(* IEC 61131-3 sources: SRCI/RobotLibrary/Library/Functions/Convert/TO_STRING (part 3) *)

(* ---- TELEGRAM_STATE_TO_STRING.st ---- *)
FUNCTION TELEGRAM_STATE_TO_STRING : STRING
// -------------------------------------------------------------------------
//  SRCI Robot Library
// -------------------------------------------------------------------------
//
//  Object:      TelegramStateToString
//  Author:      Thorsten Brach
//  Date:        2024-11-16
//
//  Description:
//
//
//  Copyright:
//    (C) 2024 Thorsten Brach. All rights reserved
//             Licensed under the LGPL-3.0 license.
//
//  Disclaimer:
//    This project is provided without any guarantee and can be used for
//    private and commercial purposes. Any use is at the user’s
//    own risk and responsibility.
//
// -------------------------------------------------------------------------
VAR_INPUT
  /// Telegram state
  State : TelegramState;
END_VAR

  CASE State
  OF
    TelegramState.UNDEFINED                : TELEGRAM_STATE_TO_STRING := StrReplace('UNDEFINED ({0})'               ,'{0}', USINT_TO_STRING(State));
    TelegramState.ERROR_161                : TELEGRAM_STATE_TO_STRING := StrReplace('ERROR_161 ({0})'               ,'{0}', USINT_TO_STRING(State));
    TelegramState.ERROR_162                : TELEGRAM_STATE_TO_STRING := StrReplace('ERROR_162 ({0})'               ,'{0}', USINT_TO_STRING(State));
    TelegramState.ERROR_163                : TELEGRAM_STATE_TO_STRING := StrReplace('ERROR_163 ({0})'               ,'{0}', USINT_TO_STRING(State));
    TelegramState.ERROR_164                : TELEGRAM_STATE_TO_STRING := StrReplace('ERROR_164 ({0})'               ,'{0}', USINT_TO_STRING(State));
    TelegramState.ERROR_165                : TELEGRAM_STATE_TO_STRING := StrReplace('ERROR_165 ({0})'               ,'{0}', USINT_TO_STRING(State));
    TelegramState.ERROR_166                : TELEGRAM_STATE_TO_STRING := StrReplace('ERROR_166 ({0})'               ,'{0}', USINT_TO_STRING(State));
    TelegramState.ERROR_167                : TELEGRAM_STATE_TO_STRING := StrReplace('ERROR_167 ({0})'               ,'{0}', USINT_TO_STRING(State));
    TelegramState.ERROR_168                : TELEGRAM_STATE_TO_STRING := StrReplace('ERROR_168 ({0})'               ,'{0}', USINT_TO_STRING(State));
    TelegramState.ERROR_169                : TELEGRAM_STATE_TO_STRING := StrReplace('ERROR_169 ({0})'               ,'{0}', USINT_TO_STRING(State));
    TelegramState.ERROR_170                : TELEGRAM_STATE_TO_STRING := StrReplace('ERROR_170 ({0})'               ,'{0}', USINT_TO_STRING(State));
    TelegramState.ERROR_171                : TELEGRAM_STATE_TO_STRING := StrReplace('ERROR_171 ({0})'               ,'{0}', USINT_TO_STRING(State));
    TelegramState.ERROR_172                : TELEGRAM_STATE_TO_STRING := StrReplace('ERROR_172 ({0})'               ,'{0}', USINT_TO_STRING(State));
    TelegramState.ERROR_173                : TELEGRAM_STATE_TO_STRING := StrReplace('ERROR_173 ({0})'               ,'{0}', USINT_TO_STRING(State));
    TelegramState.READY_TO_RESUME          : TELEGRAM_STATE_TO_STRING := StrReplace('READY_TO_RESUME ({0})'         ,'{0}', USINT_TO_STRING(State));
    TelegramState.READY_FOR_INITIALIZATION : TELEGRAM_STATE_TO_STRING := StrReplace('READY_FOR_INITIALIZATION ({0})','{0}', USINT_TO_STRING(State));
    TelegramState.INITIALIZED              : TELEGRAM_STATE_TO_STRING := StrReplace('INITIALIZED ({0})'             ,'{0}', USINT_TO_STRING(State));
  ELSE
    TELEGRAM_STATE_TO_STRING := CONCAT('TELEGRAM_STATE_TO_STRING Function: Error -> no parsing for value ', USINT_TO_STRING(State));
  END_CASE

END_FUNCTION

(* ---- THRESHOLD_MODE_TO_STRING.st ---- *)
FUNCTION THRESHOLD_MODE_TO_STRING : STRING
// -------------------------------------------------------------------------
//  SRCI Robot Library
// -------------------------------------------------------------------------
//
//  Object:      THRESHOLD_MODE_TO_STRING
//  Author:      Thorsten Brach
//  Date:        2025-01-24
//
//  Description:
//
//
//  Copyright:
//    (C) 2025 Thorsten Brach. All rights reserved
//             Licensed under the LGPL-3.0 license.
//
//  Disclaimer:
//    This project is provided without any guarantee and can be used for
//    private and commercial purposes. Any use is at the user’s
//    own risk and responsibility.
//
// -------------------------------------------------------------------------
VAR_INPUT
  /// ThresholdMode
  Value : ThresholdMode;
END_VAR

  CASE Value
  OF
    ThresholdMode.AUTOMATIC : THRESHOLD_MODE_TO_STRING := StrReplace('AUTOMATIC ({0})','{0}' , USINT_TO_STRING(Value));
    ThresholdMode.MANUAL    : THRESHOLD_MODE_TO_STRING := StrReplace('MANUAL ({0})'   ,'{0}' , USINT_TO_STRING(Value));
  ELSE
    THRESHOLD_MODE_TO_STRING := CONCAT('THRESHOLD_MODE_TO_STRING Function: Error -> no parsing for value ', USINT_TO_STRING(Value));
  END_CASE

END_FUNCTION

(* ---- TOOL_CALCULATION_MODE_TO_STRING.st ---- *)
FUNCTION TOOL_CALCULATION_MODE_TO_STRING : STRING
// -------------------------------------------------------------------------
//  SRCI Robot Library
// -------------------------------------------------------------------------
//
//  Object:      TOOL_CALCULATION_MODE_TO_STRING
//  Author:      Thorsten Brach
//  Date:        2025-02-01
//
//  Description:
//
//
//  Copyright:
//    (C) 2025 Thorsten Brach. All rights reserved
//             Licensed under the LGPL-3.0 license.
//
//  Disclaimer:
//    This project is provided without any guarantee and can be used for
//    private and commercial purposes. Any use is at the user’s
//    own risk and responsibility.
//
// -------------------------------------------------------------------------
VAR_INPUT
  /// ToolCalculationMode
  Value : ToolCalculationMode;
END_VAR

  CASE Value
  OF
    ToolCalculationMode.TWO_POINT_Z_METHOD   : TOOL_CALCULATION_MODE_TO_STRING := StrReplace('TWO_POINT_Z_METHOD ({0})'  ,'{0}' , SINT_TO_STRING(Value));
    ToolCalculationMode.THREE_POINT_METHOD   : TOOL_CALCULATION_MODE_TO_STRING := StrReplace('THREE_POINT_METHOD ({0})'  ,'{0}' , SINT_TO_STRING(Value));
    ToolCalculationMode.FOUR_POINT_METHOD    : TOOL_CALCULATION_MODE_TO_STRING := StrReplace('FOUR_POINT_METHOD ({0})'   ,'{0}' , SINT_TO_STRING(Value));
    ToolCalculationMode.FIVE_POINT_METHOD    : TOOL_CALCULATION_MODE_TO_STRING := StrReplace('FIVE_POINT_METHOD ({0})'   ,'{0}' , SINT_TO_STRING(Value));
    ToolCalculationMode.SIX_POINT_METHOD     : TOOL_CALCULATION_MODE_TO_STRING := StrReplace('SIX_POINT_METHOD ({0})'    ,'{0}' , SINT_TO_STRING(Value));
    ToolCalculationMode.ABC_WORLD_METHOD     : TOOL_CALCULATION_MODE_TO_STRING := StrReplace('ABC_WORLD_METHOD ({0})'    ,'{0}' , SINT_TO_STRING(Value));
    ToolCalculationMode.ABC_TWO_POINT_METHOD : TOOL_CALCULATION_MODE_TO_STRING := StrReplace('ABC_TWO_POINT_METHOD ({0})','{0}' , SINT_TO_STRING(Value));
  ELSE
    TOOL_CALCULATION_MODE_TO_STRING := CONCAT('TOOL_CALCULATION_MODE_TO_STRING Function: Error -> no parsing for value ', SINT_TO_STRING(Value));
  END_CASE

END_FUNCTION

(* ---- TRAJECTORY_MODE_TO_STRING.st ---- *)
FUNCTION TRAJECTORY_MODE_TO_STRING : STRING
// -------------------------------------------------------------------------
//  SRCI Robot Library
// -------------------------------------------------------------------------
//
//  Object:      TRAJECTORY_MODE_TO_STRING
//  Author:      Thorsten Brach
//  Date:        2025-03-01
//
//  Description:
//
//
//  Copyright:
//    (C) 2025 Thorsten Brach. All rights reserved
//             Licensed under the LGPL-3.0 license.
//
//  Disclaimer:
//    This project is provided without any guarantee and can be used for
//    private and commercial purposes. Any use is at the user’s
//    own risk and responsibility.
//
// -------------------------------------------------------------------------
VAR_INPUT
  /// TrajectoryMode
  Value : TrajectoryMode;
END_VAR

  CASE Value
  OF
    TrajectoryMode.INVALID          : TRAJECTORY_MODE_TO_STRING := StrReplace('INVALID ({0})'         ,'{0}' , USINT_TO_STRING(Value));
    TrajectoryMode.LINEAR_MOVEMENT  : TRAJECTORY_MODE_TO_STRING := StrReplace('LINEAR_MOVEMENT ({0})' ,'{0}' , USINT_TO_STRING(Value));
    TrajectoryMode.PTP_MOVEMENT     : TRAJECTORY_MODE_TO_STRING := StrReplace('PTP_MOVEMENT ({0})'    ,'{0}' , USINT_TO_STRING(Value));
  ELSE
    TRAJECTORY_MODE_TO_STRING := CONCAT('TRAJECTORY_MODE_TO_STRING Function: Error -> no parsing for value ', USINT_TO_STRING(Value));
  END_CASE

END_FUNCTION

(* ---- TRANSFORM_MODE_TO_STRING.st ---- *)
FUNCTION TRANSFORM_MODE_TO_STRING : STRING
// -------------------------------------------------------------------------
//  SRCI Robot Library
// -------------------------------------------------------------------------
//
//  Object:      TRANSFORM_MODE_TO_STRING
//  Author:      Thorsten Brach
//  Date:        2025-01-24
//
//  Description:
//
//
//  Copyright:
//    (C) 2025 Thorsten Brach. All rights reserved
//             Licensed under the LGPL-3.0 license.
//
//  Disclaimer:
//    This project is provided without any guarantee and can be used for
//    private and commercial purposes. Any use is at the user’s
//    own risk and responsibility.
//
// -------------------------------------------------------------------------
VAR_INPUT
  /// TransformMode
  Value : TransformMode;
END_VAR

  CASE Value
  OF
    TransformMode.MIRROR_AT_POINT             : TRANSFORM_MODE_TO_STRING := StrReplace('MIRROR_AT_POINT ({0})'             ,'{0}' , SINT_TO_STRING(Value));
    TransformMode.MIRROR_AT_STRAIGHT_LINE     : TRANSFORM_MODE_TO_STRING := StrReplace('MIRROR_AT_STRAIGHT_LINE ({0})'     ,'{0}' , SINT_TO_STRING(Value));
    TransformMode.MIRROR_AT_PLANE             : TRANSFORM_MODE_TO_STRING := StrReplace('MIRROR_AT_PLANE ({0})'             ,'{0}' , SINT_TO_STRING(Value));
    TransformMode.ROTATE_AROUND_STRAIGHT_LINE : TRANSFORM_MODE_TO_STRING := StrReplace('ROTATE_AROUND_STRAIGHT_LINE ({0})' ,'{0}' , SINT_TO_STRING(Value));
    TransformMode.SHIFT_BY_VECTOR             : TRANSFORM_MODE_TO_STRING := StrReplace('SHIFT_BY_VECTOR ({0})'             ,'{0}' , SINT_TO_STRING(Value));
  ELSE
    TRANSFORM_MODE_TO_STRING := CONCAT('TRANSFORM_MODE_TO_STRING Function: Error -> no parsing for value ', SINT_TO_STRING(Value));
  END_CASE

END_FUNCTION

(* ---- TRIGGER_CONDITION_TO_STRING.st ---- *)
FUNCTION TRIGGER_CONDITION_TO_STRING : STRING
// -------------------------------------------------------------------------
//  SRCI Robot Library
// -------------------------------------------------------------------------
//
//  Object:      TRIGGER_CONDITION_TO_STRING
//  Author:      Thorsten Brach
//  Date:        2025-02-01
//
//  Description:
//
//
//  Copyright:
//    (C) 2025 Thorsten Brach. All rights reserved
//             Licensed under the LGPL-3.0 license.
//
//  Disclaimer:
//    This project is provided without any guarantee and can be used for
//    private and commercial purposes. Any use is at the user’s
//    own risk and responsibility.
//
// -------------------------------------------------------------------------
VAR_INPUT
  /// TriggerCondition
  Value : TriggerCondition;
END_VAR

  CASE Value
  OF
    TriggerCondition.TARGET_POSITION_TIME_MS                : TRIGGER_CONDITION_TO_STRING := StrReplace('TARGET_POSITION_TIME_MS ({0})'               ,'{0}' , SINT_TO_STRING(Value));
    TriggerCondition.TARGET_POSITION_TCP_VELOCITY_ABSOLUTE  : TRIGGER_CONDITION_TO_STRING := StrReplace('TARGET_POSITION_TCP_VELOCITY_ABSOLUTE ({0})' ,'{0}' , SINT_TO_STRING(Value));
    TriggerCondition.TARGET_POSITION_TCP_VELOCITY_PERCENT   : TRIGGER_CONDITION_TO_STRING := StrReplace('TARGET_POSITION_TCP_VELOCITY_PERCENT ({0})'  ,'{0}' , SINT_TO_STRING(Value));
    TriggerCondition.TARGET_POSITION_DISTANCE_ABSOLUTE      : TRIGGER_CONDITION_TO_STRING := StrReplace('TARGET_POSITION_DISTANCE_ABSOLUTE ({0})'     ,'{0}' , SINT_TO_STRING(Value));
    TriggerCondition.TARGET_POSITION_DISTANCE_PERCENT       : TRIGGER_CONDITION_TO_STRING := StrReplace('TARGET_POSITION_DISTANCE_PERCENT ({0})'      ,'{0}' , SINT_TO_STRING(Value));
    TriggerCondition.UNDEFINED                              : TRIGGER_CONDITION_TO_STRING := StrReplace('UNDEFINED ({0})'                             ,'{0}' , SINT_TO_STRING(Value));
    TriggerCondition.START_POSITION_DISTANCE_PERCENT        : TRIGGER_CONDITION_TO_STRING := StrReplace('START_POSITION_DISTANCE_PERCENT ({0})'       ,'{0}' , SINT_TO_STRING(Value));
    TriggerCondition.START_POSITION_DISTANCE_ABSOLUTE       : TRIGGER_CONDITION_TO_STRING := StrReplace('START_POSITION_DISTANCE_ABSOLUTE ({0})'      ,'{0}' , SINT_TO_STRING(Value));
    TriggerCondition.START_POSITION_TCP_VELOCITY_PERCENT    : TRIGGER_CONDITION_TO_STRING := StrReplace('START_POSITION_TCP_VELOCITY_PERCENT ({0})'   ,'{0}' , SINT_TO_STRING(Value));
    TriggerCondition.START_POSITION_TCP_VELOCIT_ABSOLUTE    : TRIGGER_CONDITION_TO_STRING := StrReplace('START_POSITION_TCP_VELOCIT_ABSOLUTE ({0})'   ,'{0}' , SINT_TO_STRING(Value));
    TriggerCondition.START_POSITION_TIME_MS                 : TRIGGER_CONDITION_TO_STRING := StrReplace('START_POSITION_TCP_VELOCIT_ABSOLUTE ({0})'   ,'{0}' , SINT_TO_STRING(Value));
  ELSE
    TRIGGER_CONDITION_TO_STRING := CONCAT('TRIGGER_CONDITION_TO_STRING Function: Error -> no parsing for value ', SINT_TO_STRING(Value));
  END_CASE

END_FUNCTION

(* ---- TRIGGER_MODE_IO_TO_STRING.st ---- *)
FUNCTION TRIGGER_MODE_IO_TO_STRING : STRING
// -------------------------------------------------------------------------
//  SRCI Robot Library
// -------------------------------------------------------------------------
//
//  Object:      TRIGGER_MODE_IO_TO_STRING
//  Author:      Thorsten Brach
//  Date:        2025-02-01
//
//  Description:
//
//
//  Copyright:
//    (C) 2025 Thorsten Brach. All rights reserved
//             Licensed under the LGPL-3.0 license.
//
//  Disclaimer:
//    This project is provided without any guarantee and can be used for
//    private and commercial purposes. Any use is at the user’s
//    own risk and responsibility.
//
// -------------------------------------------------------------------------
VAR_INPUT
  /// TriggerModeIo
  Value : TriggerModeIo;
END_VAR

  CASE Value
  OF
    TriggerModeIo.INVALID                                                             : TRIGGER_MODE_IO_TO_STRING := StrReplace('INVALID ({0})'                                                              ,'{0}' , SINT_TO_STRING(Value));
    TriggerModeIo.DIGITAL_INPUT_RISING_EDGE                                           : TRIGGER_MODE_IO_TO_STRING := StrReplace('DIGITAL_INPUT_RISING_EDGE ({0})'                                            ,'{0}' , SINT_TO_STRING(Value));
    TriggerModeIo.DIGITAL_INPUT_FALLING_EDGE                                          : TRIGGER_MODE_IO_TO_STRING := StrReplace('DIGITAL_INPUT_FALLING_EDGE ({0})'                                           ,'{0}' , SINT_TO_STRING(Value));
    TriggerModeIo.DIGITAL_INPUT_RISING_OR_FALLING_EDGE                                : TRIGGER_MODE_IO_TO_STRING := StrReplace('DIGITAL_INPUT_RISING_OR_FALLING_EDGE ({0})'                                 ,'{0}' , SINT_TO_STRING(Value));
    TriggerModeIo.DIGITAL_INPUT_RISING_OR_FALLING_EDGE_INVERTED                       : TRIGGER_MODE_IO_TO_STRING := StrReplace('DIGITAL_INPUT_RISING_OR_FALLING_EDGE_INVERTED ({0})'                        ,'{0}' , SINT_TO_STRING(Value));
    TriggerModeIo.DIGITAL_OUTPUT_RISING_EDGE                                          : TRIGGER_MODE_IO_TO_STRING := StrReplace('DIGITAL_OUTPUT_RISING_EDGE ({0})'                                           ,'{0}' , SINT_TO_STRING(Value));
    TriggerModeIo.DIGITAL_OUTPUT_FALLING_EDGE                                         : TRIGGER_MODE_IO_TO_STRING := StrReplace('DIGITAL_OUTPUT_FALLING_EDGE ({0})'                                          ,'{0}' , SINT_TO_STRING(Value));
    TriggerModeIo.DIGITAL_OUTPUT_RISING_OR_FALLING_EDGE                               : TRIGGER_MODE_IO_TO_STRING := StrReplace('DIGITAL_OUTPUT_RISING_OR_FALLING_EDGE ({0})'                                ,'{0}' , SINT_TO_STRING(Value));
    TriggerModeIo.DIGITAL_OUTPUT_RISING_OR_FALLING_EDGE_INVERTED                      : TRIGGER_MODE_IO_TO_STRING := StrReplace('DIGITAL_OUTPUT_RISING_OR_FALLING_EDGE_INVERTED ({0})'                       ,'{0}' , SINT_TO_STRING(Value));
    TriggerModeIo.ANALOG_INPUT_EXCEEDING_DEFINED_THRESHOLD                            : TRIGGER_MODE_IO_TO_STRING := StrReplace('ANALOG_INPUT_EXCEEDING_DEFINED_THRESHOLD ({0})'                             ,'{0}' , SINT_TO_STRING(Value));
    TriggerModeIo.ANALOG_INPUT_FALLING_BELOW_DEFINED_THRESHOLD                        : TRIGGER_MODE_IO_TO_STRING := StrReplace('ANALOG_INPUT_FALLING_BELOW_DEFINED_THRESHOLD ({0})'                         ,'{0}' , SINT_TO_STRING(Value));
    TriggerModeIo.ANALOG_INPUT_EXCEEDING_OR_FALLING_BELOW_DEFINED_THRESHOLD           : TRIGGER_MODE_IO_TO_STRING := StrReplace('ANALOG_INPUT_EXCEEDING_OR_FALLING_BELOW_DEFINED_THRESHOLD ({0})'            ,'{0}' , SINT_TO_STRING(Value));
    TriggerModeIo.ANALOG_INPUT_EXCEEDING_OR_FALLING_BELOW_DEFINED_THRESHOLD_INVERTED  : TRIGGER_MODE_IO_TO_STRING := StrReplace('ANALOG_INPUT_EXCEEDING_OR_FALLING_BELOW_DEFINED_THRESHOLD_INVERTED ({0})'   ,'{0}' , SINT_TO_STRING(Value));
    TriggerModeIo.ANALOG_INPUT_ENTERING_DEFINED_RANGE                                 : TRIGGER_MODE_IO_TO_STRING := StrReplace('ANALOG_INPUT_ENTERING_DEFINED_RANGE ({0})'                                  ,'{0}' , SINT_TO_STRING(Value));
    TriggerModeIo.ANALOG_INPUT_LEAVING_DEFINED_RANGE                                  : TRIGGER_MODE_IO_TO_STRING := StrReplace('ANALOG_INPUT_LEAVING_DEFINED_RANGE ({0})'                                   ,'{0}' , SINT_TO_STRING(Value));
    TriggerModeIo.ANALOG_INPUT_ENTERING_OR_LEAVING_DEFINED_RANGE                      : TRIGGER_MODE_IO_TO_STRING := StrReplace('ANALOG_INPUT_ENTERING_OR_LEAVING_DEFINED_RANGE ({0})'                       ,'{0}' , SINT_TO_STRING(Value));
    TriggerModeIo.ANALOG_INPUT_ENTERING_OR_LEAVING_DEFINED_RANGE_INVERTED             : TRIGGER_MODE_IO_TO_STRING := StrReplace('ANALOG_INPUT_ENTERING_OR_LEAVING_DEFINED_RANGE_INVERTED ({0})'              ,'{0}' , SINT_TO_STRING(Value));
    TriggerModeIo.ANALOG_OUTPUT_EXCEEDING_DEFINED_THRESHOLD                           : TRIGGER_MODE_IO_TO_STRING := StrReplace('ANALOG_OUTPUT_EXCEEDING_DEFINED_THRESHOLD ({0})'                            ,'{0}' , SINT_TO_STRING(Value));
    TriggerModeIo.ANALOG_OUTPUT_FALLING_BELOW_DEFINED_THRESHOLD                       : TRIGGER_MODE_IO_TO_STRING := StrReplace('ANALOG_OUTPUT_FALLING_BELOW_DEFINED_THRESHOLD ({0})'                        ,'{0}' , SINT_TO_STRING(Value));
    TriggerModeIo.ANALOG_OUTPUT_EXCEEDING_OR_FALLING_BELOW_DEFINED_THRESHOLD          : TRIGGER_MODE_IO_TO_STRING := StrReplace('ANALOG_OUTPUT_EXCEEDING_OR_FALLING_BELOW_DEFINED_THRESHOLD ({0})'           ,'{0}' , SINT_TO_STRING(Value));
    TriggerModeIo.ANALOG_OUTPUT_EXCEEDING_OR_FALLING_BELOW_DEFINED_THRESHOLD_INVERTED : TRIGGER_MODE_IO_TO_STRING := StrReplace('ANALOG_OUTPUT_EXCEEDING_OR_FALLING_BELOW_DEFINED_THRESHOLD_INVERTED ({0})'  ,'{0}' , SINT_TO_STRING(Value));
    TriggerModeIo.ANALOG_OUTPUT_ENTERING_DEFINED_RANGE                                : TRIGGER_MODE_IO_TO_STRING := StrReplace('ANALOG_OUTPUT_ENTERING_DEFINED_RANGE ({0})'                                 ,'{0}' , SINT_TO_STRING(Value));
    TriggerModeIo.ANALOG_OUTPUT_LEAVING_DEFINED_RANGE                                 : TRIGGER_MODE_IO_TO_STRING := StrReplace('ANALOG_OUTPUT_LEAVING_DEFINED_RANGE ({0})'                                  ,'{0}' , SINT_TO_STRING(Value));
    TriggerModeIo.ANALOG_OUTPUT_ENTERING_OR_LEAVING_DEFINED_RANGE                     : TRIGGER_MODE_IO_TO_STRING := StrReplace('ANALOG_OUTPUT_ENTERING_OR_LEAVING_DEFINED_RANGE ({0})'                      ,'{0}' , SINT_TO_STRING(Value));
    TriggerModeIo.ANALOG_OUTPUT_ENTERING_OR_LEAVING_DEFINED_RANGE_INVERTED            : TRIGGER_MODE_IO_TO_STRING := StrReplace('ANALOG_OUTPUT_ENTERING_OR_LEAVING_DEFINED_RANGE_INVERTED ({0})'             ,'{0}' , SINT_TO_STRING(Value));
    TriggerModeIo.INTEGER_REGISTER_EXCEEDING_DEFINED_THRESHOLD                        : TRIGGER_MODE_IO_TO_STRING := StrReplace('INTEGER_REGISTER_EXCEEDING_DEFINED_THRESHOLD ({0})'                         ,'{0}' , SINT_TO_STRING(Value));
    TriggerModeIo.INTEGER_REGISTER_FALLING_BELOW_DEFINED_THRESHOLD                    : TRIGGER_MODE_IO_TO_STRING := StrReplace('INTEGER_REGISTER_FALLING_BELOW_DEFINED_THRESHOLD ({0})'                     ,'{0}' , SINT_TO_STRING(Value));
    TriggerModeIo.INTEGER_REGISTER_EXCEEDING_OR_FALLING_BELOW_DEFINED_THRESHOLD       : TRIGGER_MODE_IO_TO_STRING := StrReplace('INTEGER_REGISTER_EXCEEDING_OR_FALLING_BELOW_DEFINED_THRESHOLD ({0})'        ,'{0}' , SINT_TO_STRING(Value));
    TriggerModeIo.INTEGER_REGISTER_EXCEEDING_OR_FALLING_BELOW_DEFINED_VALUE_INVERTED  : TRIGGER_MODE_IO_TO_STRING := StrReplace('INTEGER_REGISTER_EXCEEDING_OR_FALLING_BELOW_DEFINED_VALUE_INVERTED ({0})'   ,'{0}' , SINT_TO_STRING(Value));
    TriggerModeIo.INTEGER_REGISTER_ENTERING_DEFINED_RANGE                             : TRIGGER_MODE_IO_TO_STRING := StrReplace('INTEGER_REGISTER_ENTERING_DEFINED_RANGE ({0})'                              ,'{0}' , SINT_TO_STRING(Value));
    TriggerModeIo.INTEGER_REGISTER_LEAVING_DEFINED_RANGE                              : TRIGGER_MODE_IO_TO_STRING := StrReplace('INTEGER_REGISTER_LEAVING_DEFINED_RANGE ({0})'                               ,'{0}' , SINT_TO_STRING(Value));
    TriggerModeIo.INTEGER_REGISTER_ENTERING_OR_LEAVING_DEFINED_RANGE                  : TRIGGER_MODE_IO_TO_STRING := StrReplace('INTEGER_REGISTER_ENTERING_OR_LEAVING_DEFINED_RANGE ({0})'                   ,'{0}' , SINT_TO_STRING(Value));
    TriggerModeIo.INTEGER_REGISTER_ENTERING_OR_LEAVING_DEFINED_RANGE_INVERTED         : TRIGGER_MODE_IO_TO_STRING := StrReplace('INTEGER_REGISTER_ENTERING_OR_LEAVING_DEFINED_RANGE_INVERTED ({0})'          ,'{0}' , SINT_TO_STRING(Value));
    TriggerModeIo.REAL_REGISTER_EXCEEDING_DEFINED_THRESHOLD                           : TRIGGER_MODE_IO_TO_STRING := StrReplace('REAL_REGISTER_EXCEEDING_DEFINED_THRESHOLD ({0})'                            ,'{0}' , SINT_TO_STRING(Value));
    TriggerModeIo.REAL_REGISTER_FALLING_BELOW_DEFINED_THRESHOLD                       : TRIGGER_MODE_IO_TO_STRING := StrReplace('REAL_REGISTER_FALLING_BELOW_DEFINED_THRESHOLD ({0})'                        ,'{0}' , SINT_TO_STRING(Value));
    TriggerModeIo.REAL_REGISTER_EXCEEDING_OR_FALLING_BELOW_DEFINED_THRESHOLD          : TRIGGER_MODE_IO_TO_STRING := StrReplace('REAL_REGISTER_EXCEEDING_OR_FALLING_BELOW_DEFINED_THRESHOLD ({0})'           ,'{0}' , SINT_TO_STRING(Value));
    TriggerModeIo.REAL_REGISTER_EXCEEDING_OR_FALLING_BELOW_DEFINED_THRESHOLD_INVERTED : TRIGGER_MODE_IO_TO_STRING := StrReplace('REAL_REGISTER_EXCEEDING_OR_FALLING_BELOW_DEFINED_THRESHOLD_INVERTED ({0})'  ,'{0}' , SINT_TO_STRING(Value));
    TriggerModeIo.REAL_REGISTER_ENTERING_DEFINED_RANGE                                : TRIGGER_MODE_IO_TO_STRING := StrReplace('REAL_REGISTER_ENTERING_DEFINED_RANGE ({0})'                                 ,'{0}' , SINT_TO_STRING(Value));
    TriggerModeIo.REAL_REGISTER_LEAVING_DEFINED_RANGE                                 : TRIGGER_MODE_IO_TO_STRING := StrReplace('REAL_REGISTER_LEAVING_DEFINED_RANGE ({0})'                                  ,'{0}' , SINT_TO_STRING(Value));
    TriggerModeIo.REAL_REGISTER_ENTERING_OR_LEAVING_DEFINED_RANGE                     : TRIGGER_MODE_IO_TO_STRING := StrReplace('REAL_REGISTER_ENTERING_OR_LEAVING_DEFINED_RANGE ({0})'                      ,'{0}' , SINT_TO_STRING(Value));
    TriggerModeIo.REAL_REGISTER_ENTERING_OR_LEAVING_DEFINED_RANGE_INVERTED            : TRIGGER_MODE_IO_TO_STRING := StrReplace('REAL_REGISTER_ENTERING_OR_LEAVING_DEFINED_RANGE_INVERTED ({0})'             ,'{0}' , SINT_TO_STRING(Value));
  ELSE
    TRIGGER_MODE_IO_TO_STRING := CONCAT('TRIGGER_MODE_IO_TO_STRING Function: Error -> no parsing for value ', SINT_TO_STRING(Value));
  END_CASE

END_FUNCTION

(* ---- TRIGGER_MODE_LIMIT_TO_STRING.st ---- *)
FUNCTION TRIGGER_MODE_LIMIT_TO_STRING : STRING
// -------------------------------------------------------------------------
//  SRCI Robot Library
// -------------------------------------------------------------------------
//
//  Object:      TRIGGER_MODE_LIMIT_TO_STRING
//  Author:      Thorsten Brach
//  Date:        2025-03-02
//
//  Description:
//
//
//  Copyright:
//    (C) 2025 Thorsten Brach. All rights reserved
//             Licensed under the LGPL-3.0 license.
//
//  Disclaimer:
//    This project is provided without any guarantee and can be used for
//    private and commercial purposes. Any use is at the user’s
//    own risk and responsibility.
//
// -------------------------------------------------------------------------
VAR_INPUT
  /// TriggerModeLimit
  Value : TriggerModeLimit;
END_VAR

  CASE Value
  OF
    TriggerModeLimit.INVALID         : TRIGGER_MODE_LIMIT_TO_STRING := StrReplace('INVALID ({0})'         ,'{0}' , SINT_TO_STRING(Value));
    TriggerModeLimit.JOINT_CURRENT   : TRIGGER_MODE_LIMIT_TO_STRING := StrReplace('JOINT_CURRENT ({0})'   ,'{0}' , SINT_TO_STRING(Value));
    TriggerModeLimit.FORCE           : TRIGGER_MODE_LIMIT_TO_STRING := StrReplace('FORCE ({0})'           ,'{0}' , SINT_TO_STRING(Value));
    TriggerModeLimit.FOLLOWING_ERROR : TRIGGER_MODE_LIMIT_TO_STRING := StrReplace('FOLLOWING_ERROR ({0})' ,'{0}' , SINT_TO_STRING(Value));
    TriggerModeLimit.TEMPERATURE     : TRIGGER_MODE_LIMIT_TO_STRING := StrReplace('TEMPERATURE ({0})'     ,'{0}' , SINT_TO_STRING(Value));
  ELSE
    TRIGGER_MODE_LIMIT_TO_STRING := CONCAT('TRIGGER_MODE_LIMIT_TO_STRING Function: Error -> no parsing for value ', SINT_TO_STRING(Value));
  END_CASE

END_FUNCTION

(* ---- TRIGGER_MODE_MEASUREMENT_TO_STRING.st ---- *)
FUNCTION TRIGGER_MODE_MEASUREMENT_TO_STRING : STRING
// -------------------------------------------------------------------------
//  SRCI Robot Library
// -------------------------------------------------------------------------
//
//  Object:      TRIGGER_MODE_MEASUREMENT_TO_STRING
//  Author:      Thorsten Brach
//  Date:        2025-01-24
//
//  Description:
//
//
//  Copyright:
//    (C) 2025 Thorsten Brach. All rights reserved
//             Licensed under the LGPL-3.0 license.
//
//  Disclaimer:
//    This project is provided without any guarantee and can be used for
//    private and commercial purposes. Any use is at the user’s
//    own risk and responsibility.
//
// -------------------------------------------------------------------------
VAR_INPUT
  /// TriggerMode
  Value : TriggerModeMeasurement;
END_VAR

  CASE Value
  OF
    TriggerModeMeasurement.NO_TRIGGER                   : TRIGGER_MODE_MEASUREMENT_TO_STRING := StrReplace('NO_TRIGGER ({0})'                   ,'{0}' , USINT_TO_STRING(Value));
    TriggerModeMeasurement.POSITIVE_START_NEGATIVE_STOP : TRIGGER_MODE_MEASUREMENT_TO_STRING := StrReplace('POSITIVE_START_NEGATIVE_STOP ({0})' ,'{0}' , USINT_TO_STRING(Value));
    TriggerModeMeasurement.POSITIVE_START_STOP          : TRIGGER_MODE_MEASUREMENT_TO_STRING := StrReplace('POSITIVE_START_STOP ({0})'          ,'{0}' , USINT_TO_STRING(Value));
  ELSE
    TRIGGER_MODE_MEASUREMENT_TO_STRING := CONCAT('TRIGGER_MODE_MEASUREMENT_TO_STRING Function: Error -> no parsing for value ', USINT_TO_STRING(Value));
  END_CASE

END_FUNCTION

(* ---- TRIGGER_REACTION_MODE_TO_STRING.st ---- *)
FUNCTION TRIGGER_REACTION_MODE_TO_STRING : STRING
// -------------------------------------------------------------------------
//  SRCI Robot Library
// -------------------------------------------------------------------------
//
//  Object:      TRIGGER_REACTION_MODE_TO_STRING
//  Author:      Thorsten Brach
//  Date:        2025-02-01
//
//  Description:
//
//
//  Copyright:
//    (C) 2025 Thorsten Brach. All rights reserved
//             Licensed under the LGPL-3.0 license.
//
//  Disclaimer:
//    This project is provided without any guarantee and can be used for
//    private and commercial purposes. Any use is at the user’s
//    own risk and responsibility.
//
// -------------------------------------------------------------------------
VAR_INPUT
  /// TriggerReactionMode
  Value : TriggerReactionMode;
END_VAR

  CASE Value
  OF

    TriggerReactionMode.NO_REACTION                : TRIGGER_REACTION_MODE_TO_STRING := StrReplace('NO_REACTION ({0})'                 ,'{0}' , SINT_TO_STRING(Value));
    TriggerReactionMode.INTERRUPT                  : TRIGGER_REACTION_MODE_TO_STRING := StrReplace('INTERRUPT ({0})'                   ,'{0}' , SINT_TO_STRING(Value));
    TriggerReactionMode.GROUP_STOP                 : TRIGGER_REACTION_MODE_TO_STRING := StrReplace('GROUP_STOP ({0})'                  ,'{0}' , SINT_TO_STRING(Value));
    TriggerReactionMode.DISABLE_ROBOT              : TRIGGER_REACTION_MODE_TO_STRING := StrReplace('DISABLE_ROBOT ({0})'               ,'{0}' , SINT_TO_STRING(Value));
    TriggerReactionMode.STOP_ACTUAL_MOTION_COMMAND : TRIGGER_REACTION_MODE_TO_STRING := StrReplace('STOP_ACTUAL_MOTION_COMMAND ({0})'  ,'{0}' , SINT_TO_STRING(Value));
  ELSE
    TRIGGER_REACTION_MODE_TO_STRING := CONCAT('TRIGGER_REACTION_MODE_TO_STRING Function: Error -> no parsing for value ', SINT_TO_STRING(Value));
  END_CASE

END_FUNCTION

(* ---- TURN_MODE_TO_STRING.st ---- *)
FUNCTION TURN_MODE_TO_STRING : STRING
// -------------------------------------------------------------------------
//  SRCI Robot Library
// -------------------------------------------------------------------------
//
//  Object:      TURN_MODE_TO_STRING
//  Author:      Thorsten Brach
//  Date:        2025-01-23
//
//  Description:
//
//
//  Copyright:
//    (C) 2025 Thorsten Brach. All rights reserved
//             Licensed under the LGPL-3.0 license.
//
//  Disclaimer:
//    This project is provided without any guarantee and can be used for
//    private and commercial purposes. Any use is at the user’s
//    own risk and responsibility.
//
// -------------------------------------------------------------------------
VAR_INPUT
  /// TurnMode
  Value : TurnMode;
END_VAR

  CASE Value
  OF
    TurnMode.USE_TURN_NUMBER : TURN_MODE_TO_STRING := StrReplace('USE_TURN_NUMBER ({0})','{0}' , USINT_TO_STRING(Value));
    TurnMode.SAME            : TURN_MODE_TO_STRING := StrReplace('SAME ({0})'           ,'{0}' , USINT_TO_STRING(Value));
    TurnMode.FREE            : TURN_MODE_TO_STRING := StrReplace('FREE ({0})'           ,'{0}' , USINT_TO_STRING(Value));
  ELSE
    TURN_MODE_TO_STRING := CONCAT('TURN_MODE_TO_STRING Function: Error -> no parsing for value ', USINT_TO_STRING(Value));
  END_CASE

END_FUNCTION

(* ---- UNIT_LIMIT_AXIS_TO_STRING.st ---- *)
FUNCTION UNIT_LIMIT_AXIS_TO_STRING : STRING
// -------------------------------------------------------------------------
//  SRCI Robot Library
// -------------------------------------------------------------------------
//
//  Object:      ORI_MODE_TO_STRING
//  Author:      Thorsten Brach
//  Date:        2025-02-25
//
//  Description:
//
//
//  Copyright:
//    (C) 2025 Thorsten Brach. All rights reserved
//             Licensed under the LGPL-3.0 license.
//
//  Disclaimer:
//    This project is provided without any guarantee and can be used for
//    private and commercial purposes. Any use is at the user’s
//    own risk and responsibility.
//
// -------------------------------------------------------------------------
VAR_INPUT
  /// UnitLimitAxis
  Value : UnitLimitAxis;
END_VAR

  CASE Value
  OF
    UnitLimitAxis.PERCENTAGE  : UNIT_LIMIT_AXIS_TO_STRING := StrReplace('PERCENTAGE ({0})'  ,'{0}' , USINT_TO_STRING(Value));
    UnitLimitAxis.NEWTONMETER : UNIT_LIMIT_AXIS_TO_STRING := StrReplace('NEWTONMETER ({0})' ,'{0}' , USINT_TO_STRING(Value));
    UnitLimitAxis.MILLIAMPERE : UNIT_LIMIT_AXIS_TO_STRING := StrReplace('MILLIAMPERE ({0})' ,'{0}' , USINT_TO_STRING(Value));
  ELSE
    UNIT_LIMIT_AXIS_TO_STRING := CONCAT('UNIT_LIMIT_AXIS_TO_STRING Function: Error -> no parsing for value ', USINT_TO_STRING(Value));
  END_CASE

END_FUNCTION

(* ---- VALID_REAL_TO_STRING.st ---- *)
FUNCTION VALID_REAL_TO_STRING : STRING
// -------------------------------------------------------------------------
//  SRCI Robot Library
// -------------------------------------------------------------------------
//
//  Object:      VALID_REAL_TO_STRING
//  Author:      Thorsten Brach
//  Date:        2025-02-26
//
//  Description:
//
//
//  Copyright:
//    (C) 2025 Thorsten Brach. All rights reserved
//             Licensed under the LGPL-3.0 license.
//
//  Disclaimer:
//    This project is provided without any guarantee and can be used for
//    private and commercial purposes. Any use is at the user’s
//    own risk and responsibility.
//
// -------------------------------------------------------------------------
VAR_INPUT
  /// Real
  Value : REAL;
END_VAR

  IF ( SysDepIsValidReal(Value))
  THEN
    VALID_REAL_TO_STRING := REAL_TO_STRING(Value);
  ELSE
    VALID_REAL_TO_STRING := 'NaN';
  END_IF

END_FUNCTION

(* ---- WORD_TO_STRING_BIN.st ---- *)
FUNCTION WORD_TO_STRING_BIN : STRING
// -------------------------------------------------------------------------
//  SRCI Robot Library
// -------------------------------------------------------------------------
//
//  Object:      WORD_TO_STRING_BIN
//  Author:      Thorsten Brach
//  Date:        2025-02-03
//
//  Description:
//    Converts a BYTE to a STRING with binary notation
//
//  Copyright:
//    (C) 2024 Thorsten Brach. All rights reserved
//             Licensed under the LGPL-3.0 license.
//
//  Disclaimer:
//    This project is provided without any guarantee and can be used for
//    private and commercial purposes. Any use is at the user’s
//    own risk and responsibility.
//
// -------------------------------------------------------------------------
VAR_INPUT
 /// Value to convert
 Value : WORD;
END_VAR

  WORD_TO_STRING_BIN := '2#';

  IF (Value.15)
  THEN
    WORD_TO_STRING_BIN := CONCAT(WORD_TO_STRING_BIN, '1');
  ELSE
    WORD_TO_STRING_BIN := CONCAT(WORD_TO_STRING_BIN, '0');
  END_IF

  IF (Value.14)
  THEN
    WORD_TO_STRING_BIN := CONCAT(WORD_TO_STRING_BIN, '1');
  ELSE
    WORD_TO_STRING_BIN := CONCAT(WORD_TO_STRING_BIN, '0');
  END_IF

  IF (Value.13)
  THEN
    WORD_TO_STRING_BIN := CONCAT(WORD_TO_STRING_BIN, '1');
  ELSE
    WORD_TO_STRING_BIN := CONCAT(WORD_TO_STRING_BIN, '0');
  END_IF

  IF (Value.12)
  THEN
    WORD_TO_STRING_BIN := CONCAT(WORD_TO_STRING_BIN, '1_');
  ELSE
    WORD_TO_STRING_BIN := CONCAT(WORD_TO_STRING_BIN, '0_');
  END_IF

  IF (Value.11)
  THEN
    WORD_TO_STRING_BIN := CONCAT(WORD_TO_STRING_BIN, '1');
  ELSE
    WORD_TO_STRING_BIN := CONCAT(WORD_TO_STRING_BIN, '0');
  END_IF

  IF (Value.10)
  THEN
    WORD_TO_STRING_BIN := CONCAT(WORD_TO_STRING_BIN, '1');
  ELSE
    WORD_TO_STRING_BIN := CONCAT(WORD_TO_STRING_BIN, '0');
  END_IF

  IF (Value.09)
  THEN
    WORD_TO_STRING_BIN := CONCAT(WORD_TO_STRING_BIN, '1');
  ELSE
    WORD_TO_STRING_BIN := CONCAT(WORD_TO_STRING_BIN, '0');
  END_IF

  IF (Value.08)
  THEN
    WORD_TO_STRING_BIN := CONCAT(WORD_TO_STRING_BIN, '1_');
  ELSE
    WORD_TO_STRING_BIN := CONCAT(WORD_TO_STRING_BIN, '0_');
  END_IF

  IF (Value.7)
  THEN
    WORD_TO_STRING_BIN := CONCAT(WORD_TO_STRING_BIN, '1');
  ELSE
    WORD_TO_STRING_BIN := CONCAT(WORD_TO_STRING_BIN, '0');
  END_IF

  IF (Value.6)
  THEN
    WORD_TO_STRING_BIN := CONCAT(WORD_TO_STRING_BIN, '1');
  ELSE
    WORD_TO_STRING_BIN := CONCAT(WORD_TO_STRING_BIN, '0');
  END_IF

  IF (Value.5)
  THEN
    WORD_TO_STRING_BIN := CONCAT(WORD_TO_STRING_BIN, '1');
  ELSE
    WORD_TO_STRING_BIN := CONCAT(WORD_TO_STRING_BIN, '0');
  END_IF

  IF (Value.4)
  THEN
    WORD_TO_STRING_BIN := CONCAT(WORD_TO_STRING_BIN, '1_');
  ELSE
    WORD_TO_STRING_BIN := CONCAT(WORD_TO_STRING_BIN, '0_');
  END_IF

  IF (Value.3)
  THEN
    WORD_TO_STRING_BIN := CONCAT(WORD_TO_STRING_BIN, '1');
  ELSE
    WORD_TO_STRING_BIN := CONCAT(WORD_TO_STRING_BIN, '0');
  END_IF

  IF (Value.2)
  THEN
    WORD_TO_STRING_BIN := CONCAT(WORD_TO_STRING_BIN, '1');
  ELSE
    WORD_TO_STRING_BIN := CONCAT(WORD_TO_STRING_BIN, '0');
  END_IF

  IF (Value.1)
  THEN
    WORD_TO_STRING_BIN := CONCAT(WORD_TO_STRING_BIN, '1');
  ELSE
    WORD_TO_STRING_BIN := CONCAT(WORD_TO_STRING_BIN, '0');
  END_IF

  IF (Value.0)
  THEN
    WORD_TO_STRING_BIN := CONCAT(WORD_TO_STRING_BIN, '1');
  ELSE
    WORD_TO_STRING_BIN := CONCAT(WORD_TO_STRING_BIN, '0');
  END_IF

  WORD_TO_STRING_BIN := CONCAT(WORD_TO_STRING_BIN, ' (');
  WORD_TO_STRING_BIN := CONCAT(WORD_TO_STRING_BIN, WORD_TO_STRING(Value));
  WORD_TO_STRING_BIN := CONCAT(WORD_TO_STRING_BIN, ')');

END_FUNCTION

(* ---- WORK_AREA_REACTION_MODE_TO_STRING.st ---- *)
FUNCTION WORK_AREA_REACTION_MODE_TO_STRING : STRING
// -------------------------------------------------------------------------
//  SRCI Robot Library
// -------------------------------------------------------------------------
//
//  Object:      WORK_AREA_REACTION_MODE_TO_STRING
//  Author:      Thorsten Brach
//  Date:        2025-02-01
//
//  Description:
//
//
//  Copyright:
//    (C) 2025 Thorsten Brach. All rights reserved
//             Licensed under the LGPL-3.0 license.
//
//  Disclaimer:
//    This project is provided without any guarantee and can be used for
//    private and commercial purposes. Any use is at the user’s
//    own risk and responsibility.
//
// -------------------------------------------------------------------------
VAR_INPUT
  /// WorkAreaReactionMode
  Value : WorkAreaReactionMode;
END_VAR

  CASE Value
  OF
    WorkAreaReactionMode.NO_REACTION : WORK_AREA_REACTION_MODE_TO_STRING := StrReplace('NO_REACTION ({0})','{0}' , USINT_TO_STRING(Value));
    WorkAreaReactionMode.ABORT       : WORK_AREA_REACTION_MODE_TO_STRING := StrReplace('ABORT ({0})'      ,'{0}' , USINT_TO_STRING(Value));
    WorkAreaReactionMode.INTERRUPT   : WORK_AREA_REACTION_MODE_TO_STRING := StrReplace('INTERRUPT ({0})'  ,'{0}' , USINT_TO_STRING(Value));
  ELSE
    WORK_AREA_REACTION_MODE_TO_STRING := CONCAT('WORK_AREA_REACTION_MODE_TO_STRING Function: Error -> no parsing for value ', USINT_TO_STRING(Value));
  END_CASE

END_FUNCTION

(* ---- WORK_AREA_REACTIONMODE_TO_STRING.st ---- *)
FUNCTION WORK_AREA_REACTIONMODE_TO_STRING : STRING
// -------------------------------------------------------------------------
//  SRCI Robot Library
// -------------------------------------------------------------------------
//
//  Object:      WORK_AREA_REACTIONMODE_TO_STRING
//  Author:      Thorsten Brach
//  Date:        2025-02-01
//
//  Description:
//
//
//  Copyright:
//    (C) 2025 Thorsten Brach. All rights reserved
//             Licensed under the LGPL-3.0 license.
//
//  Disclaimer:
//    This project is provided without any guarantee and can be used for
//    private and commercial purposes. Any use is at the user’s
//    own risk and responsibility.
//
// -------------------------------------------------------------------------
VAR_INPUT
  /// WorkAreaReactionMode
  Value : WorkAreaReactionMode;
END_VAR

  CASE Value
  OF

    WorkAreaReactionMode.NO_REACTION : StrReplace('NO_REACTION ({0})','{0}' , USINT_TO_STRING(Value));
    WorkAreaReactionMode.ABORT       : StrReplace('ABORT ({0})'      ,'{0}' , USINT_TO_STRING(Value));
    WorkAreaReactionMode.INTERRUPT   : StrReplace('INTERRUPT ({0})'  ,'{0}' , USINT_TO_STRING(Value));

  END_CASE

END_FUNCTION
